(* IEC 61131-3 sources: Std_PalletMover/Class/Hal_Lidar_Base, 1 file *)

(* ---- Hal_Lidar_Base.st ---- *)
#Define MAXBEAMS 2750 // 275° * 10 beams = 0.1 beam per Degree

(*!
<Class
	Name               = "Hal_Lidar_Base"
	Revision           = "0.0"
	RealtimeTask       = "false"
	CyclicTask         = "false"
	BackgroundTask     = "true"
	Sigmatek           = "false"
	OSInterface        = "false"
	HighPriority       = "false"
	Automatic          = "false"
	UpdateMode         = "Prescan"
	SharedCommandTable = "true"
	Objectsize         = "(284,120)">
	<Channels>
		<Server Name="ClassSvr" Visualized="false" Initialize="false" WriteProtected="true" Retentive="false"/>
		<Server Name="Direction" Visualized="false" Initialize="false" WriteProtected="false" Retentive="SRam"/>
		<Server Name="ScannerPosition" Visualized="false" Initialize="false" WriteProtected="false" Retentive="SRam"/>
	</Channels>
</Class>
*)
Hal_Lidar_Base : CLASS
	TYPE
	  eDirection :  //! <Type Public="true" Name="eDirection"/>
	  (
	    d_Fwd,
	    d_Bwd
	  )$UDINT;
	  eScannerPosition :  //! <Type Public="true" Name="eScannerPosition"/>
	  (
	    sp_LeftCorner,
	    sp_Middle,
	    sp_RightCorner
	  )$UDINT;
	  tData : DINT;
#pragma pack(push, 1)
	  tScanFieldStatus : STRUCT  //! <Type Public="true" Name="tScanFieldStatus"/>
	    sfs_WarningFieldDetection : DINT;
	    sfs_StopFieldDetection : DINT;
	    sfs_EStopFieldDetection : DINT;
	  END_STRUCT;
#pragma pack(pop)
#pragma pack(push, 1)
	  tVisuData : STRUCT  //! <Type Public="true" Name="tVisuData"/>
	    vd_Direction : Hal_Lidar_Base::eDirection;
	    vd_StartRange : DINT;
	    vd_EndRange : DINT;
	    vd_nrOfBeams : DINT;
	    vd_Beams : ARRAY [1..MAXBEAMS] OF UINT;
	  END_STRUCT;
#pragma pack(pop)
	END_TYPE
  //Servers:
	ClassSvr 	: SvrChCmd_DINT;
	ScannerPosition 	: SvrCh_eScannerPosition_PTofCls_Hal_Lidar_Base;
	Direction 	: SvrCh_eDirection_PTofCls_Hal_Lidar_Base;
  //Clients:
  //Variables:
  //Functions:

	FUNCTION VIRTUAL GLOBAL Background
		VAR_INPUT
			EAX 	: UDINT;
		END_VAR
		VAR_OUTPUT
			state (EAX) 	: UDINT := READY;
		END_VAR;

	FUNCTION VIRTUAL GLOBAL GetVisuData
		VAR_OUTPUT
			retValue 	: tVisuData;
		END_VAR;

	FUNCTION VIRTUAL GLOBAL GetLidarInfo;

	FUNCTION VIRTUAL GLOBAL GetScannerData
		VAR_OUTPUT
			retValue 	: tScanFieldStatus;
		END_VAR;
  //Tables:
	FUNCTION @STD
		VAR_OUTPUT
			ret_code	: CONFSTATES;
		END_VAR;
	FUNCTION GLOBAL TAB @CT_;
END_CLASS;

FUNCTION VIRTUAL GLOBAL Hal_Lidar_Base::GetVisuData
  #pragma warning(disable: 73);
  #pragma warning(disable: 76);
  VAR_OUTPUT
		retValue 	: tVisuData;
	END_VAR

  #pragma warning(default: 73);
  #pragma warning(default: 76);

END_FUNCTION

FUNCTION VIRTUAL GLOBAL Hal_Lidar_Base::GetLidarInfo

END_FUNCTION

FUNCTION VIRTUAL GLOBAL Hal_Lidar_Base::Background
	VAR_INPUT
		EAX 	: UDINT;
	END_VAR
	VAR_OUTPUT
		state (EAX) 	: UDINT;(* := READY *)
	END_VAR

END_FUNCTION

FUNCTION VIRTUAL GLOBAL Hal_Lidar_Base::GetScannerData
	#pragma warning(disable: 73);
  #pragma warning(disable: 76);
  VAR_OUTPUT
		retValue 	: tScanFieldStatus;
	END_VAR

  #pragma warning(default: 73);
  #pragma warning(default: 76);

END_FUNCTION
